// TwinCAT 3 PLC project MemRingBufferExample
// ProgramVersion: 3.1.4026.20
// libraries:
//   Tc2_Standard, * (Beckhoff Automation GmbH)
//   Tc2_System, * (Beckhoff Automation GmbH)
//   Tc2_Utilities, * (Beckhoff Automation GmbH)
//   Tc3_Interfaces, * (Beckhoff Automation GmbH)
//   Tc3_Module, * (Beckhoff Automation GmbH)
// project tree:
//   DUTs/ ST_DataSetEntry.TcDUT (not stored)
//   GVLs/ GVL.TcGVL (not stored)
//   POUs/ FB_DataSetFifo.TcPOU (not stored), MAIN.TcPOU
//   / Standard.TcTTO (not stored)

// ---- POUs/MAIN.TcPOU
PROGRAM MAIN
VAR
	fbFifo 		: FB_DataSetFifo := ( bOverwrite := TRUE );
	newEntry	: ST_DataSetEntry;
	oldEntry	: ST_DataSetEntry;
	bSuccess	: BOOL;
	nCount		: UDINT;
	nLoad		: UDINT;

	bReset 		: BOOL := TRUE;
	bAdd 		: BOOL := TRUE;
	bGet		: BOOL := TRUE;
	bRemove		: BOOL := TRUE;
END_VAR

IF bReset THEN
	bReset := FALSE;
	(* reset fifo (clear all entries) *)
	fbFifo.A_Reset(	in := newEntry, bOk=>bSuccess, nCount=> nCount, nLoad => nLoad );
END_IF

IF bAdd THEN
	bAdd := FALSE;

	(* create new or modify data set entry *)
	newEntry.bFlag := NOT newEntry.bFlag;
	newEntry.nValue := newEntry.nValue + 1;
	newEntry.sMsg := BYTE_TO_STRING(newEntry.nValue);

	(* add new entry to the fifo *)
	fbFifo.A_Add(	in := newEntry, bOk=>bSuccess, nCount=> nCount, nLoad => nLoad );
END_IF

IF bGet THEN
	bGet := FALSE;
	(* get (but not delete) oldest entry *)
	fbFifo.A_Get( out => oldEntry, bOk => bSuccess, nCount => nCount, nLoad => nLoad );
END_IF

IF bRemove THEN
	bRemove:= FALSE;
	(* remove oldest entry *)
	fbFifo.A_Remove( out => oldEntry, bOk => bSuccess, nCount => nCount, nLoad => nLoad );
END_IF

END_PROGRAM
